FUNCTION_BLOCK Mc3MoveVelocityTask EXTENDS Mc3MotionTask
VAR
	_TargetVelocity : LREAL;
	McMoveVelocity	: ARRAY[0..1] OF Tc3_Mc3Ptp.MC_MoveVelocity;
	Active			: UDINT;
	_McBufferMode	: Tc3_Mc3Ptp.EBufferMode;
END_VAR

PROPERTY BufferMode : REFERENCE TO Tc3_Mc3Ptp.EBufferMode
GET
BufferMode REF= _McBufferMode;
END_GET
END_PROPERTY

{attribute 'monitoring' := 'call'}
PROPERTY Busy : BOOL
GET
Busy := McMoveVelocity[Active].Busy;
END_GET
END_PROPERTY

METHOD CyclicLogic
VAR
    i : UDINT;
END_VAR
FOR i := 0 TO 1 DO
	McMoveVelocity[i](Axis		   := _Axis.Axis,
					  Velocity	   := _TargetVelocity,
					  Acceleration := _Axis.Acceleration,
					  Deceleration := _Axis.Deceleration,
					  Jerk		   := _Axis.Jerk,
					  BufferMode   := _McBufferMode);

	McMoveVelocity[i].Execute := FALSE;
END_FOR
END_METHOD

{attribute 'monitoring' := 'call'}
PROPERTY Error : BOOL
GET
Error := McMoveVelocity[Active].Error;
END_GET
END_PROPERTY

{attribute 'monitoring' := 'call'}
PROPERTY ErrorId : UDINT
GET
ErrorID := McMoveVelocity[Active].ErrorID;
END_GET
END_PROPERTY

METHOD Execute : BOOL;
IF Active = 0 THEN
	Active := 1;
	McMoveVelocity[Active](Axis			:= _Axis.Axis,
						   Execute		:= TRUE,
						   Velocity		:= _TargetVelocity,
						   Acceleration := _Axis.Acceleration,
						   Deceleration := _Axis.Deceleration,
						   Jerk			:= _Axis.Jerk,
						   BufferMode	:= _McBufferMode);
ELSE
	Active := 0;
	McMoveVelocity[Active](Axis			:= _Axis.Axis,
						   Execute		:= TRUE,
						   Velocity		:= _TargetVelocity,
						   Acceleration := _Axis.Acceleration,
						   Deceleration := _Axis.Deceleration,
						   Jerk			:= _Axis.Jerk,
						   BufferMode	:= _McBufferMode);
END_IF

Execute := TRUE;
END_METHOD

{attribute 'monitoring' := 'call'}
PROPERTY TargetVelocity : LREAL
SET
_TargetVelocity := TargetVelocity;
END_SET
END_PROPERTY

END_FUNCTION_BLOCK

(* stored: Version 1.1.0.1, ProductVersion 3.1.4026.20
   POU Mc3MoveVelocityTask: Id {bd0ee06a-1e66-4837-b725-c224e7aaf68d}, SpecialFunc None
   Property BufferMode: Id {f74642bb-089f-402f-8387-a6f849c14a62}
   Get Get: Id {6c3c0fb4-a0a1-4b4f-a361-d1796eee54bc}
   Property Busy: Id {27d9f99d-4462-4176-b47b-e317a6ba89f0}
   Get Get: Id {b620416b-1da0-4fa8-a1ff-53d750bb82b4}
   Method CyclicLogic: Id {bdb743f2-ef4b-49f3-804c-a677508d205b}
   Property Error: Id {381002b5-441c-4515-8220-8743cb85c337}
   Get Get: Id {d3686b92-700d-4d05-bb18-2f30db4633e2}
   Property ErrorId: Id {7c202154-dbf2-4e35-bd42-4e774339c1f2}
   Get Get: Id {893ba4fe-3687-4387-b8ef-3426a423c3d7}
   Method Execute: Id {ca421f7d-254d-4a03-aba1-a0d508c8a55b}
   Property TargetVelocity: Id {a4e5d071-c12a-4223-9567-78281b54abb7}
   Set Set: Id {f4da5916-4516-420b-9949-cec2340759db} *)
